FUNCTION_BLOCK FB_Transfer
VAR_INPUT
	nLine					: INT;
	fTimer_Comb				: REAL;
	fTimer_Clip				: REAL;
	fTimer_Move_Comb		: REAL;
END_VAR
VAR_OUTPUT
	nDoneTransfer			: INT;
	bDoneTransfer			: BOOL;
END_VAR
VAR
	fbCylinder_Comb			: FB_Cylinder;
	fbCylinder_Clip			: FB_Cylinder;
	fbCylinder_Move_Comb	: FB_Cylinder;
	// ===== SIM COMPONENTS ==============
	fbCylinderSim_Comb		: FB_Cylinder_Sim;
	fbCylinderSim_Clip		: FB_Cylinder_Sim;
	fbCylinderSim_Move_Comb	: FB_Cylinder_Sim;
	// ===== INTERFACES ==================
	iCylinder_Comb			: I_Cylinder;
	iCylinder_Clip			: I_Cylinder;
	iCylinder_Move_Comb		: I_Cylinder;
	//====== VAR MOTHOD ==================
	nState					: INT;
	nStateEnable			: INT;
	nState_Reset			: INT;
	tTimer_Reset			: TON;
	fbTimer_Comb			: TON;
	fbTimer_Clip			: TON;
	fbTimer_Move_Comb		: TON;
	//======== VAR HMI Transfer Setting ====
END_VAR

IF bSimMode THEN
	iCylinder_Clip 	:= fbCylinderSim_Clip;
	fbCylinderSim_Clip();
	iCylinder_Comb	:= fbCylinderSim_Comb;
	fbCylinderSim_Comb();
	iCylinder_Move_Comb	:= fbCylinderSim_Move_Comb;
	fbCylinderSim_Move_Comb();
ELSE
	iCylinder_Clip 	:= fbCylinder_Clip;
	fbCylinder_Clip(id := 1);
	iCylinder_Comb	:= fbCylinder_Comb;
	fbCylinder_Comb(id := 1);
	iCylinder_Move_Comb	:= fbCylinder_Move_Comb;
	fbCylinder_Move_Comb(id := 1);
END_IF

METHOD Auto : BOOL
VAR_INPUT
END_VAR
fbTimer_Clip(PT := REAL_TO_TIME(fTimer_Clip)*1000);
fbTimer_Comb(PT := REAL_TO_TIME(fTimer_Comb)*1000);
fbTimer_Move_Comb(PT := REAL_TO_TIME(fTimer_Move_Comb)*1000);
CASE nState OF 
	0: // init value
		Auto		:= FALSE;
		fbTimer_Move_Comb(IN := FALSE);
		fbTimer_Clip(IN	:= FALSE);
		fbTimer_Comb(IN	:= FALSE);
		nState		:= 1;
	1: // Cylinder Clip and Comb Extend hold cup
		bDoneTransfer 	:= FALSE;
		iCylinder_Clip.Extend();
		iCylinder_Comb.Extend();
		fbTimer_Clip(IN	:= TRUE);
		fbTimer_Comb(IN	:= TRUE);
		IF iCylinder_Clip.bIsExtend AND iCylinder_Comb.bIsExtend THEN
			nState	:= 2;
		ELSIF fbTimer_Comb.Q AND NOT fbTimer_Clip.Q THEN
			IF nLine = 1 THEN
				F_SetError(18,nLine := 1);
			ELSIF nLine = 2 THEN
				F_SetError(40,nLine := 2);
			END_IF
		ELSIF fbTimer_Clip.Q AND NOT fbTimer_Comb.Q THEN
			IF nLine = 1 THEN
				F_SetError(20,nLine := 1);
			ELSIF nLine = 2 THEN
				F_SetError(42,nLine := 2);
			END_IF
		ELSIF iCylinder_Clip.bIsExtend AND fbTimer_Comb.Q THEN
			IF nLine = 1 THEN
				F_SetError(18,nLine := 1);
			ELSIF nLine = 2 THEN
				F_SetError(40,nLine := 2);
			END_IF
		ELSIF iCylinder_Comb.bIsExtend AND fbTimer_Clip.Q THEN
			IF nLine = 1 THEN
				F_SetError(20,nLine := 1);
			ELSIF nLine = 2 THEN
				F_SetError(42,nLine := 2);
			END_IF
		ELSIF fbTimer_Comb.Q AND fbTimer_Clip.Q THEN
			IF nLine = 1 THEN
				F_SetError(18,nLine := 1);
			ELSIF nLine = 2 THEN
				F_SetError(40,nLine := 2);
			END_IF
		END_IF
	2: // Cylinder_Move_Comb Extend move cup
		fbTimer_Clip(IN	:= FALSE);
		fbTimer_Comb(IN	:= FALSE);
		fbTimer_Move_Comb(IN := TRUE);
		iCylinder_Move_Comb.Extend();
		IF iCylinder_Move_Comb.bIsExtend THEN
			nState	:= 3;
		ELSIF fbTimer_Move_Comb.Q THEN
			IF nLine = 1 THEN
				F_SetError(22,nLine := 1);
			ELSIF nLine = 2 THEN
				F_SetError(44,nLine := 2);
			END_IF
		END_IF
	3: // retract clip and comb
		fbTimer_Comb(IN := TRUE);
		fbTimer_Move_Comb(IN := FALSE);
		iCylinder_Comb.Retract();
		IF iCylinder_Comb.bIsRetract THEN
			nState	:= 33;
		ELSIF fbTimer_Comb.Q THEN
			IF nLine = 1 THEN
				F_SetError(17,nLine := 1);
			ELSIF nLine = 2 THEN
				F_SetError(39,nLine := 2);
			END_IF
		END_IF
	33:
		fbTimer_Clip(IN := TRUE);
		fbTimer_Comb(IN := FALSE);
		iCylinder_Clip.Retract();
		IF iCylinder_Clip.bIsRetract THEN
			nDoneTransfer	:= nDoneTransfer + 1;
			bDoneTransfer 	:= TRUE;
			IF nLine = 1 THEN 
				bToDropcup1			:= TRUE;
			ELSIF nLine = 2 THEN
				bToDropcup2			:= TRUE;
			END_IF
			IF nDoneTransfer > 8 THEN
				nDoneTransfer := 8;
			END_IF
			nState	:= 4;
		ELSIF fbTimer_Clip.Q THEN
			IF nLine = 1 THEN
				F_SetError(19,nLine := 1);
			ELSIF nLine = 2 THEN
				F_SetError(41,nLine := 2);
			END_IF
		END_IF
	4://Move_Comb Retract
		fbTimer_Clip(IN := FALSE);
		fbTimer_Move_Comb(IN := TRUE);
		iCylinder_Move_Comb.Retract();
		IF iCylinder_Move_Comb.bIsRetract THEN
			nState	:= 5;
		ELSIF fbTimer_Move_Comb.Q THEN
			IF nLine = 1 THEN
				F_SetError(21,nLine := 1);
			ELSIF nLine = 2 THEN
				F_SetError(43,nLine := 2);
			END_IF
		END_IF
	5:// Complete
		fbTimer_Move_Comb(IN := FALSE);
		Auto		:= TRUE;
		nState		:= 0;	
END_CASE
END_METHOD

METHOD Enable : BOOL
VAR_INPUT
END_VAR
fbTimer_Clip(PT := REAL_TO_TIME(fTimer_Clip)*1000);
fbTimer_Comb(PT := REAL_TO_TIME(fTimer_Comb)*1000);
fbTimer_Move_Comb(PT := REAL_TO_TIME(fTimer_Move_Comb)*1000);
CASE nStateEnable OF
	0:// init 
		Enable					:= FALSE;
		fbTimer_Clip(IN	:= FALSE);
		fbTimer_Comb(IN	:= FALSE);
		fbTimer_Move_Comb(IN := FALSE);
		nStateEnable			:= 1;
	1:// Retract Comb and Clip
		iCylinder_Clip.Retract();
		iCylinder_Comb.Retract();
		fbTimer_Clip(IN	:= TRUE);
		fbTimer_Comb(IN	:= TRUE);
		IF iCylinder_Clip.bIsRetract AND iCylinder_Comb.bIsRetract THEN
			nStateEnable		:= 2;
		ELSIF fbTimer_Clip.Q AND NOT fbTimer_Comb.Q THEN
			nStateEnable		:= 10;
		ELSIF fbTimer_Comb.Q AND NOT fbTimer_Clip.Q THEN
			nStateEnable		:= 11;
		END_IF	
	2:// Retract MoveComb
		fbTimer_Clip(IN	:= FALSE);
		fbTimer_Comb(IN	:= FALSE);
		iCylinder_Move_Comb.Retract();
		fbTimer_Move_Comb.IN	:= TRUE;
		IF iCylinder_Move_Comb.bIsRetract THEN
			nStateEnable		:= 3;
		ELSIF fbTimer_Move_Comb.Q THEN
			nState				:= 12;
		END_IF
	3:// Enable
		fbTimer_Move_Comb(IN := FALSE);
		Enable					:= TRUE;
	10:// Error Cylinder Clip
		IF nLine = 1 THEN
			F_SetError(17,nLine := 1);
			nState	:= 99;
		ELSIF nLine = 2 THEN
			F_SetError(35,nLine := 2);
			nState	:= 99;
		END_IF
	11:// Error Cylinder Comb
		IF nLine = 1 THEN
			F_SetError(16,nLine := 1);
			nState	:= 99;
		ELSIF nLine = 2 THEN
			F_SetError(34,nLine := 2);
			nState	:= 99;
		END_IF
	12:// Error Cylinder MoveComb
		IF nLine = 1 THEN
			F_SetError(18,nLine := 1);
			nState	:= 99;
		ELSIF nLine = 2 THEN
			F_SetError(36,nLine := 2);
			nState	:= 99;
		END_IF
	99:// Error
END_CASE
END_METHOD

METHOD Init : BOOL
VAR_INPUT
END_VAR
nState		 := 0;
nStateEnable := 0;
bDoneTransfer := FALSE;
nDoneTransfer := 0;
END_METHOD

METHOD Manual : BOOL
VAR_INPUT
	bCylinder_Comb_Extend			: BOOL;
	bCylinder_Comb_Retract			: BOOL;
	bCylinder_Clip_Extend			: BOOL;
	bCylinder_Clip_Retract			: BOOL;
	bCylinder_Move_Comb_Extend		: BOOL;
	bCylinder_Move_Comb_Retract		: BOOL;
END_VAR
IF bCylinder_Comb_Extend THEN
	iCylinder_Comb.Extend();
	IF iCylinder_Comb.bIsExtend THEN
		fbTimer_Comb(IN := FALSE);
	ELSE
		fbTimer_Comb(PT := REAL_TO_TIME(fTimer_Comb)*1000);
			IF fbTimer_Comb.Q THEN
				IF nLine = 1 THEN
					F_SetError(18,nLine := 1);
				ELSIF nLine = 2 THEN
					F_SetError(40,nLine := 2);
				END_IF
			END_IF
	END_IF
END_IF

IF bCylinder_Comb_Retract THEN
	iCylinder_Comb.Retract();
	IF iCylinder_Comb.bIsRetract THEN
		fbTimer_Comb(IN := FALSE);
	ELSE
		fbTimer_Comb(PT := REAL_TO_TIME(fTimer_Comb)*1000);
			IF fbTimer_Comb.Q THEN
				IF nLine = 1 THEN
					F_SetError(17,nLine := 1);
				ELSIF nLine = 2 THEN
					F_SetError(39,nLine := 2);
				END_IF
			END_IF
	END_IF
END_IF

IF bCylinder_Clip_Extend THEN
	iCylinder_Clip.Extend();
	IF iCylinder_Clip.bIsExtend THEN
		fbTimer_Clip(IN := FALSE);
	ELSE
		fbTimer_Clip(PT := REAL_TO_TIME(fTimer_Clip)*1000);
			IF fbTimer_Clip.Q THEN
				IF nLine = 1 THEN
					F_SetError(20,nLine := 1);
				ELSIF nLine = 2 THEN
					F_SetError(42,nLine := 2);
				END_IF
			END_IF
	END_IF
END_IF


IF bCylinder_Clip_Retract THEN
	iCylinder_Clip.Retract();	
	IF iCylinder_Clip.bIsRetract THEN
		fbTimer_Clip(IN := FALSE);
	ELSE
		fbTimer_Clip(PT := REAL_TO_TIME(fTimer_Clip)*1000);
			IF fbTimer_Clip.Q THEN
				IF nLine = 1 THEN
					F_SetError(19,nLine := 1);
				ELSIF nLine = 2 THEN
					F_SetError(41,nLine := 2);
				END_IF
			END_IF
	END_IF
END_IF

IF bCylinder_Move_Comb_Extend THEN
	iCylinder_Move_Comb.Extend();
	IF iCylinder_Move_Comb.bIsExtend THEN
		fbTimer_Move_Comb(IN := FALSE);
	ELSE
		fbTimer_Move_Comb(PT := REAL_TO_TIME(fTimer_Move_Comb)*1000);
			IF fbTimer_Move_Comb.Q THEN
				IF nLine = 1 THEN
					F_SetError(22,nLine := 1);
				ELSIF nLine = 2 THEN
					F_SetError(44,nLine := 2);
				END_IF
			END_IF
	END_IF
END_IF

IF bCylinder_Move_Comb_Retract THEN
	iCylinder_Move_Comb.Retract();
	IF iCylinder_Move_Comb.bIsRetract THEN
		fbTimer_Move_Comb(IN := FALSE);
	ELSE
		fbTimer_Move_Comb(PT := REAL_TO_TIME(fTimer_Move_Comb)*1000);
			IF fbTimer_Move_Comb.Q THEN
				IF nLine = 1 THEN
					F_SetError(21,nLine := 1);
				ELSIF nLine = 2 THEN
					F_SetError(43,nLine := 2);
				END_IF
			END_IF
	END_IF
END_IF
END_METHOD

METHOD Reset : BOOL
VAR_INPUT
END_VAR
iCylinder_Clip.Retract();
fbTimer_Clip(IN	:= FALSE);
fbTimer_Comb(IN	:= FALSE);
fbTimer_Move_Comb(IN := FALSE);

CASE nState_Reset OF
	0:
		iCylinder_Comb.Retract();
		tTimer_Reset(IN := TRUE, PT := T#300MS);
		IF tTimer_Reset.Q OR iCylinder_Comb.bIsRetract THEN
			nState_Reset := 1;
		END_IF
	1:
		iCylinder_Move_Comb.Retract();
		nState_Reset := 0;
END_CASE
END_METHOD

METHOD Stop : BOOL
VAR_INPUT
END_VAR
fbTimer_Clip(IN	:= FALSE);
fbTimer_Comb(IN	:= FALSE);
fbTimer_Move_Comb(IN := FALSE);
END_METHOD

END_FUNCTION_BLOCK

(* stored: Version 1.1.0.1, ProductVersion 3.1.4024.12
   POU FB_Transfer: Id {18dc2db3-5ecd-4211-80b1-8da0d86e8f52}, SpecialFunc None
   Method Auto: Id {a18e3b75-c925-4aab-bb01-50e79f209c3d}
   Method Enable: Id {d751481a-6f77-432e-bcda-c667c2a94dd0}
   Method Init: Id {ace05526-e93a-48fb-b372-82c4543adae8}
   Method Manual: Id {f0c3f1b0-2965-4a71-87a8-d99df85f8ed8}
   Method Reset: Id {5ffa7dd5-079f-4576-92a2-bcc40e8754a6}
   Method Stop: Id {baec0fc2-6e50-43ca-b136-2da2a4544107} *)
